// TwinCAT 3 PLC project Main
// ProgramVersion: 3.1.4023.0
// libraries:
//   Tc2_Standard, * (Beckhoff Automation GmbH)
//   Tc2_System, * (Beckhoff Automation GmbH)
//   Tc3_Module, * (Beckhoff Automation GmbH)
// project tree:
//   / PlcTask.TcTTO
//   POUs/ FB_FinalTest.TcPOU, MAIN.TcPOU
// real-time tasks:
//   TASK PlcTask: cycle T#10ms, priority 20, ADS port 350
// I/O:
//   DEVICE Device 1 (TC3 EIP Adapter), AmsNetId 10.100.103.242.2.1
//     Box 1 (TC EtherNet/IP Slave)

CONFIGURATION Main
    RESOURCE PLC ON TwinCAT3
        TASK PlcTask(INTERVAL := T#10ms, PRIORITY := 20);
        PROGRAM MAIN WITH PlcTask : MAIN;
    END_RESOURCE
END_CONFIGURATION

// ---- POUs/MAIN.TcPOU
PROGRAM MAIN
VAR
	bChange : BOOL := TRUE;
	
END_VAR

END_PROGRAM

// ---- POUs/FB_FinalTest.TcPOU
FUNCTION_BLOCK PUBLIC FB_FinalTest

VAR
	
END_VAR

METHOD FB_Opto22Read : BOOL
VAR_INPUT
END_VAR
END_METHOD

METHOD FB_Opto22Write : BOOL
VAR_INPUT
END_VAR
END_METHOD

METHOD PUBLIC LeakTest : BOOL
VAR_INPUT
END_VAR
END_METHOD

METHOD PRIVATE ModuleCheck : BOOL
VAR_INPUT
END_VAR
END_METHOD

END_FUNCTION_BLOCK
